Fanuc KAREL source: ke00001.KL

-- PROVISIONAL review KL for V940-1; original PC SHA256 a172d607428fd7650a3de53d3facc16d04480bc2f10096c8a991740ff5dde4ef
-- Incomplete behavior may be omitted. Consult companion uncertainty JSON. Do not deploy.
PROGRAM KE00001
%NOLOCKGROUP
BEGIN
  -- V9_ZERO_TABLE_METADATA_HINT layout=0002_ascii; no indexed target words; source/name/runtime held
  -- UNRESOLVED_PC offsets 5-12; opcodes 9D,23
  -- UNRESOLVED_PC offsets 17-41; opcodes 27,22,22,2A,22,31
  -- UNRESOLVED_PC offsets 46-50; opcodes 7F
END KE00001
